// TIA Portal V21 export
FUNCTION "BOWIE" : Void   // FC7, LAD
{ S7_Optimized_Access := 'TRUE' }
// stored: SetENOAutomatically false
   VAR_TEMP
      START : Bool;
   END_VAR
   VAR_TEMP   // added for the SCL form of the ladder/FBD networks
      _w1 : Bool;
      _w2 : Bool;
      _w3 : Bool;
      _w4 : Bool;
   END_VAR
BEGIN

REGION Network 1
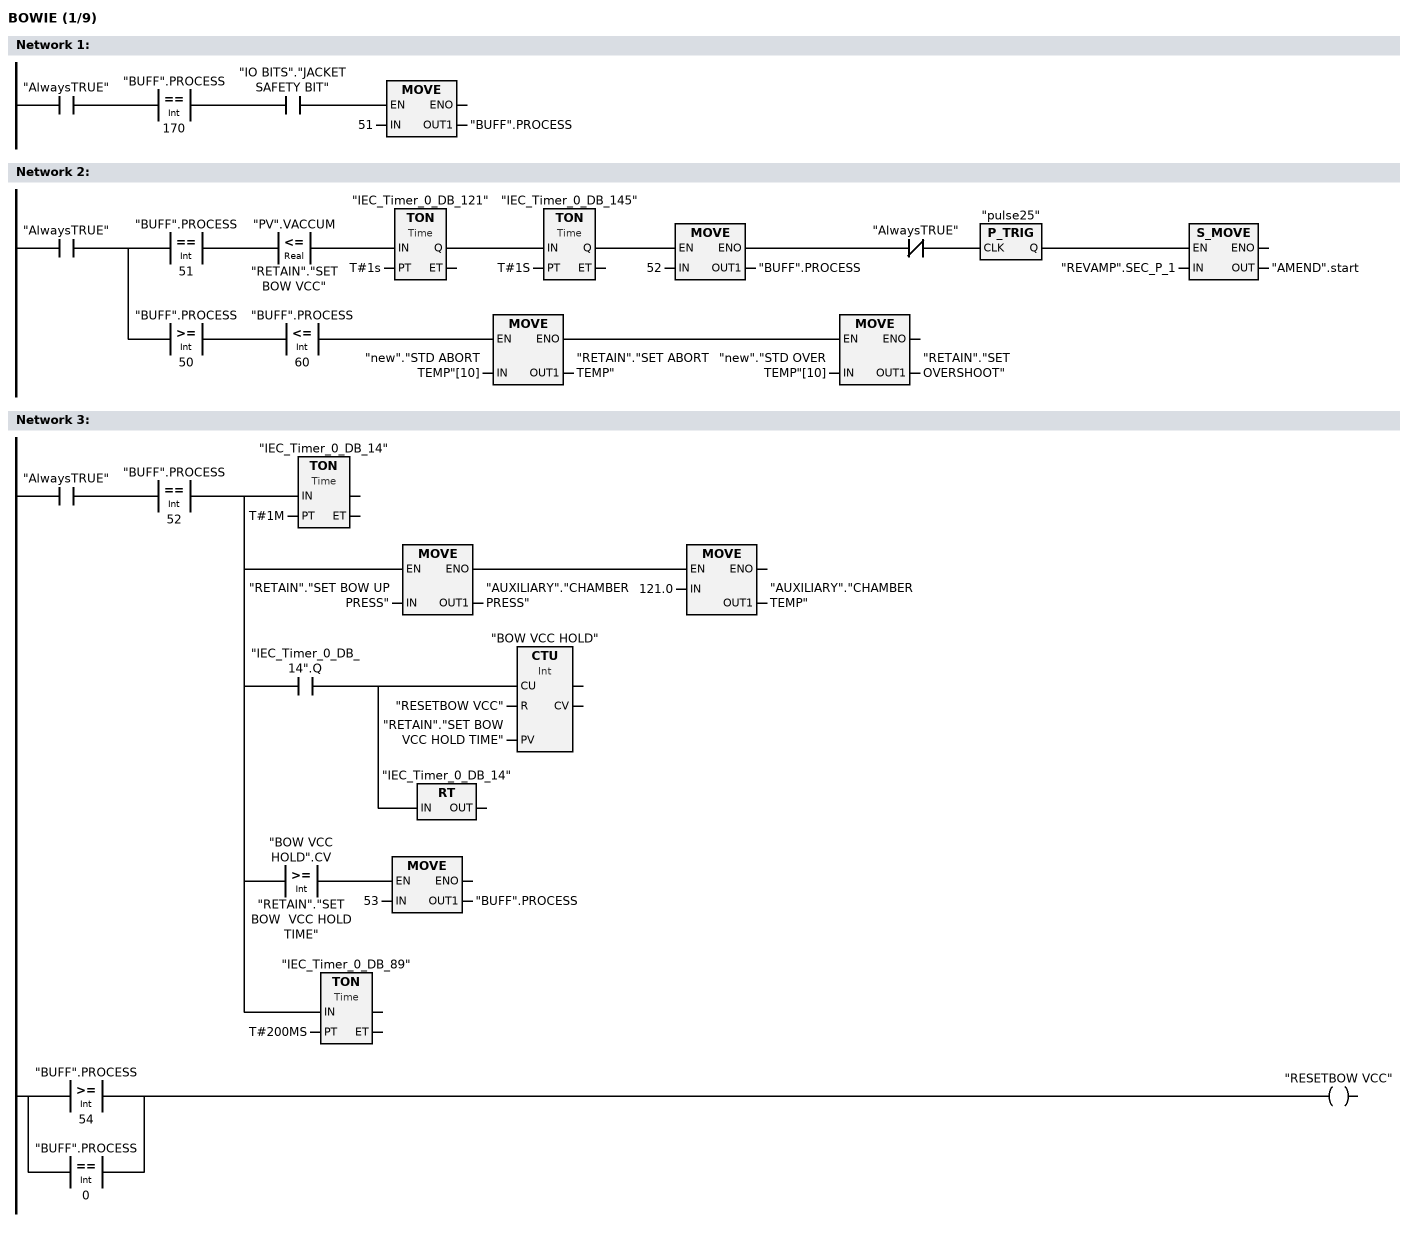
   RUNG wire#powerrail
      Contact( "AlwaysTRUE" )
      { S7_Templates := "SrcType := Int" } EQ_Contact(in1 := "BUFF".PROCESS, in2 := 170)
      Contact( "IO BITS"."JACKET SAFETY BIT" )
      Move(in := 51, out1 => "BUFF".PROCESS)
   END_RUNG
   // the same network as SCL:
   IF "AlwaysTRUE" AND ("BUFF".PROCESS = 170) AND "IO BITS"."JACKET SAFETY BIT" THEN
       "BUFF".PROCESS := 51;
   END_IF;
END_REGION

REGION Network 2
   RUNG wire#powerrail
      Contact( "AlwaysTRUE" )
      wire#w1
      { S7_Templates := "SrcType := Int" } EQ_Contact(in1 := "BUFF".PROCESS, in2 := 51)
      { S7_Templates := "SrcType := Real" } LE_Contact(in1 := "PV".VACCUM, in2 := "RETAIN"."SET BOW VCC")
      { S7_Templates := "time_type := Time" } "IEC_Timer_0_DB_121".TON(pt := T#1s, et =>)
      { S7_Templates := "time_type := Time" } "IEC_Timer_0_DB_145".TON(pt := T#1S, et =>)
      Move(in := 52, out1 => "BUFF".PROCESS)
      I_Contact( "AlwaysTRUE" )
      P_Trig( "pulse25" )
      S_Move(in := "REVAMP".SEC_P_1, out => "AMEND".start)
   END_RUNG
   RUNG wire#w1
      { S7_Templates := "SrcType := Int" } GE_Contact(in1 := "BUFF".PROCESS, in2 := 50)
      { S7_Templates := "SrcType := Int" } LE_Contact(in1 := "BUFF".PROCESS, in2 := 60)
      Move(in := "new"."STD ABORT TEMP"[10], out1 => "RETAIN"."SET ABORT TEMP")
      Move(in := "new"."STD OVER TEMP"[10], out1 => "RETAIN"."SET OVERSHOOT")
   END_RUNG
   // the same network as SCL:
   "IEC_Timer_0_DB_121".TON(IN := "AlwaysTRUE" AND ("BUFF".PROCESS = 51) AND ("PV".VACCUM <= "RETAIN"."SET BOW VCC"),
                           PT := T#1s);
   "IEC_Timer_0_DB_145".TON(IN := "IEC_Timer_0_DB_121".Q, PT := T#1S);
   IF "IEC_Timer_0_DB_145".Q THEN "BUFF".PROCESS := 52; END_IF;
   #_w1 := "IEC_Timer_0_DB_145".Q AND NOT "AlwaysTRUE";
   #_w2 := #_w1 AND NOT "pulse25";   // rising edge
   "pulse25" := #_w1;
   IF #_w2 THEN "AMEND".start := "REVAMP".SEC_P_1; END_IF;
   IF "AlwaysTRUE" AND ("BUFF".PROCESS >= 50) AND ("BUFF".PROCESS <= 60) THEN
       "RETAIN"."SET ABORT TEMP" := "new"."STD ABORT TEMP"[10];
       "RETAIN"."SET OVERSHOOT" := "new"."STD OVER TEMP"[10];
   END_IF;
END_REGION

REGION Network 3
   RUNG wire#powerrail
      Contact( "AlwaysTRUE" )
      { S7_Templates := "SrcType := Int" } EQ_Contact(in1 := "BUFF".PROCESS, in2 := 52)
      wire#w1
      { S7_Templates := "time_type := Time" } "IEC_Timer_0_DB_14".TON(pt := T#1M, et =>)
   END_RUNG
   RUNG wire#w1
      Move(in := "RETAIN"."SET BOW UP PRESS", out1 => "AUXILIARY"."CHAMBER PRESS")
      Move(in := 121.0, out1 => "AUXILIARY"."CHAMBER TEMP")
   END_RUNG
   RUNG wire#w1
      Contact( "IEC_Timer_0_DB_14".Q )
      wire#w2
      { S7_Templates := "value_type := Int" } "BOW VCC HOLD".CTU(r := "RESETBOW VCC", pv := "RETAIN"."SET BOW  VCC HOLD TIME", cv =>)
   END_RUNG
   RUNG wire#w2
      RT_Coil( "IEC_Timer_0_DB_14" )
   END_RUNG
   RUNG wire#w1
      { S7_Templates := "SrcType := Int" } GE_Contact(in1 := "BOW VCC HOLD".CV, in2 := "RETAIN"."SET BOW  VCC HOLD TIME")
      Move(in := 53, out1 => "BUFF".PROCESS)
   END_RUNG
   RUNG wire#w1
      { S7_Templates := "time_type := Time" } "IEC_Timer_0_DB_89".TON(pt := T#200MS, et =>)
   END_RUNG
   RUNG wire#powerrail
      { S7_Templates := "SrcType := Int" } GE_Contact(in1 := "BUFF".PROCESS, in2 := 54)
      wire#w3
      Coil( "RESETBOW VCC" )
   END_RUNG
   RUNG wire#powerrail
      { S7_Templates := "SrcType := Int" } EQ_Contact(in1 := "BUFF".PROCESS, in2 := 0)
   END_RUNG wire#w3
   // the same network as SCL:
   #_w1 := "AlwaysTRUE" AND ("BUFF".PROCESS = 52);
   "IEC_Timer_0_DB_14".TON(IN := #_w1, PT := T#1M);
   IF #_w1 THEN
       "AUXILIARY"."CHAMBER PRESS" := "RETAIN"."SET BOW UP PRESS";
       "AUXILIARY"."CHAMBER TEMP" := 121.0;
   END_IF;
   #_w2 := #_w1 AND "IEC_Timer_0_DB_14".Q;
   "BOW VCC HOLD".CTU(CU := #_w2, R := "RESETBOW VCC", PV := "RETAIN"."SET BOW  VCC HOLD TIME");
   IF #_w2 THEN RESET_TIMER("IEC_Timer_0_DB_14"); END_IF;
   IF #_w1 AND ("BOW VCC HOLD".CV >= "RETAIN"."SET BOW  VCC HOLD TIME") THEN "BUFF".PROCESS := 53; END_IF;
   "IEC_Timer_0_DB_89".TON(IN := #_w1, PT := T#200MS);
   "RESETBOW VCC" := ("BUFF".PROCESS >= 54) OR ("BUFF".PROCESS = 0);
END_REGION

REGION Network 4
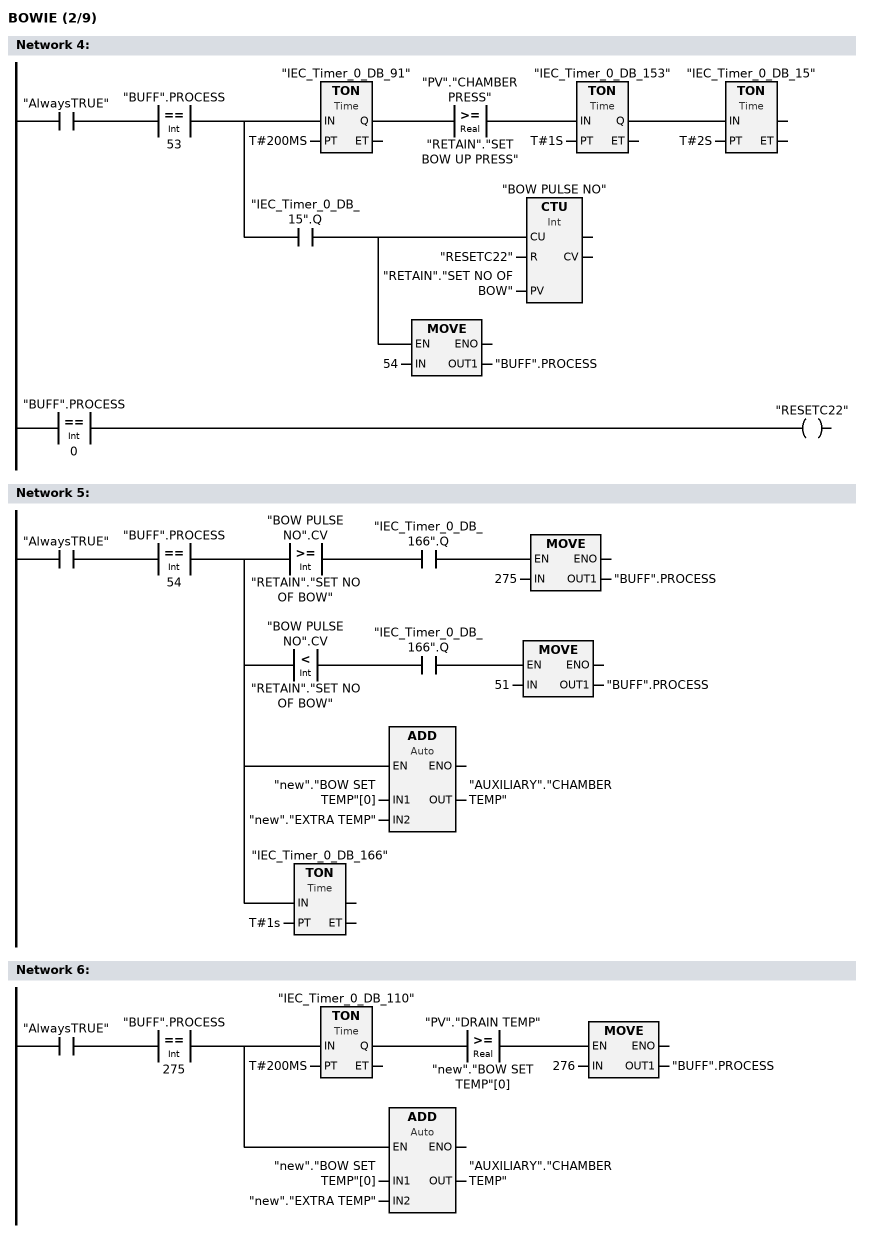
   RUNG wire#powerrail
      Contact( "AlwaysTRUE" )
      { S7_Templates := "SrcType := Int" } EQ_Contact(in1 := "BUFF".PROCESS, in2 := 53)
      wire#w1
      { S7_Templates := "time_type := Time" } "IEC_Timer_0_DB_91".TON(pt := T#200MS, et =>)
      { S7_Templates := "SrcType := Real" } GE_Contact(in1 := "PV"."CHAMBER PRESS", in2 := "RETAIN"."SET BOW UP PRESS")
      { S7_Templates := "time_type := Time" } "IEC_Timer_0_DB_153".TON(pt := T#1S, et =>)
      { S7_Templates := "time_type := Time" } "IEC_Timer_0_DB_15".TON(pt := T#2S, et =>)
   END_RUNG
   RUNG wire#w1
      Contact( "IEC_Timer_0_DB_15".Q )
      wire#w2
      { S7_Templates := "value_type := Int" } "BOW PULSE NO".CTU(r := "RESETC22", pv := "RETAIN"."SET NO OF BOW", cv =>)
   END_RUNG
   RUNG wire#w2
      Move(in := 54, out1 => "BUFF".PROCESS)
   END_RUNG
   RUNG wire#powerrail
      { S7_Templates := "SrcType := Int" } EQ_Contact(in1 := "BUFF".PROCESS, in2 := 0)
      Coil( "RESETC22" )
   END_RUNG
   // the same network as SCL:
   #_w1 := "AlwaysTRUE" AND ("BUFF".PROCESS = 53);
   "IEC_Timer_0_DB_91".TON(IN := #_w1, PT := T#200MS);
   "IEC_Timer_0_DB_153".TON(IN := "IEC_Timer_0_DB_91".Q AND ("PV"."CHAMBER PRESS" >= "RETAIN"."SET BOW UP PRESS"),
                           PT := T#1S);
   "IEC_Timer_0_DB_15".TON(IN := "IEC_Timer_0_DB_153".Q, PT := T#2S);
   #_w2 := #_w1 AND "IEC_Timer_0_DB_15".Q;
   "BOW PULSE NO".CTU(CU := #_w2, R := "RESETC22", PV := "RETAIN"."SET NO OF BOW");
   IF #_w2 THEN "BUFF".PROCESS := 54; END_IF;
   "RESETC22" := "BUFF".PROCESS = 0;
END_REGION

REGION Network 5
   RUNG wire#powerrail
      Contact( "AlwaysTRUE" )
      { S7_Templates := "SrcType := Int" } EQ_Contact(in1 := "BUFF".PROCESS, in2 := 54)
      wire#w1
      { S7_Templates := "SrcType := Int" } GE_Contact(in1 := "BOW PULSE NO".CV, in2 := "RETAIN"."SET NO OF BOW")
      Contact( "IEC_Timer_0_DB_166".Q )
      Move(in := 275, out1 => "BUFF".PROCESS)
   END_RUNG
   RUNG wire#w1
      { S7_Templates := "SrcType := Int" } LT_Contact(in1 := "BOW PULSE NO".CV, in2 := "RETAIN"."SET NO OF BOW")
      Contact( "IEC_Timer_0_DB_166".Q )
      Move(in := 51, out1 => "BUFF".PROCESS)
   END_RUNG
   RUNG wire#w1
      Add(in1 := "new"."BOW SET TEMP"[0], in2 := "new"."EXTRA TEMP", out => "AUXILIARY"."CHAMBER TEMP")
   END_RUNG
   RUNG wire#w1
      { S7_Templates := "time_type := Time" } "IEC_Timer_0_DB_166".TON(pt := T#1s, et =>)
   END_RUNG
   // the same network as SCL:
   #_w1 := "AlwaysTRUE" AND ("BUFF".PROCESS = 54);
   IF #_w1 AND ("BOW PULSE NO".CV >= "RETAIN"."SET NO OF BOW") AND "IEC_Timer_0_DB_166".Q THEN
       "BUFF".PROCESS := 275;
   END_IF;
   IF #_w1 AND ("BOW PULSE NO".CV < "RETAIN"."SET NO OF BOW") AND "IEC_Timer_0_DB_166".Q THEN
       "BUFF".PROCESS := 51;
   END_IF;
   IF #_w1 THEN "AUXILIARY"."CHAMBER TEMP" := "new"."BOW SET TEMP"[0] + "new"."EXTRA TEMP"; END_IF;
   "IEC_Timer_0_DB_166".TON(IN := #_w1, PT := T#1s);
END_REGION

REGION Network 6
   RUNG wire#powerrail
      Contact( "AlwaysTRUE" )
      { S7_Templates := "SrcType := Int" } EQ_Contact(in1 := "BUFF".PROCESS, in2 := 275)
      wire#w1
      { S7_Templates := "time_type := Time" } "IEC_Timer_0_DB_110".TON(pt := T#200MS, et =>)
      { S7_Templates := "SrcType := Real" } GE_Contact(in1 := "PV"."DRAIN TEMP", in2 := "new"."BOW SET TEMP"[0])
      Move(in := 276, out1 => "BUFF".PROCESS)
   END_RUNG
   RUNG wire#w1
      Add(in1 := "new"."BOW SET TEMP"[0], in2 := "new"."EXTRA TEMP", out => "AUXILIARY"."CHAMBER TEMP")
   END_RUNG
   // the same network as SCL:
   #_w1 := "AlwaysTRUE" AND ("BUFF".PROCESS = 275);
   "IEC_Timer_0_DB_110".TON(IN := #_w1, PT := T#200MS);
   IF "IEC_Timer_0_DB_110".Q AND ("PV"."DRAIN TEMP" >= "new"."BOW SET TEMP"[0]) THEN
       "BUFF".PROCESS := 276;
   END_IF;
   IF #_w1 THEN "AUXILIARY"."CHAMBER TEMP" := "new"."BOW SET TEMP"[0] + "new"."EXTRA TEMP"; END_IF;
END_REGION

REGION Network 7
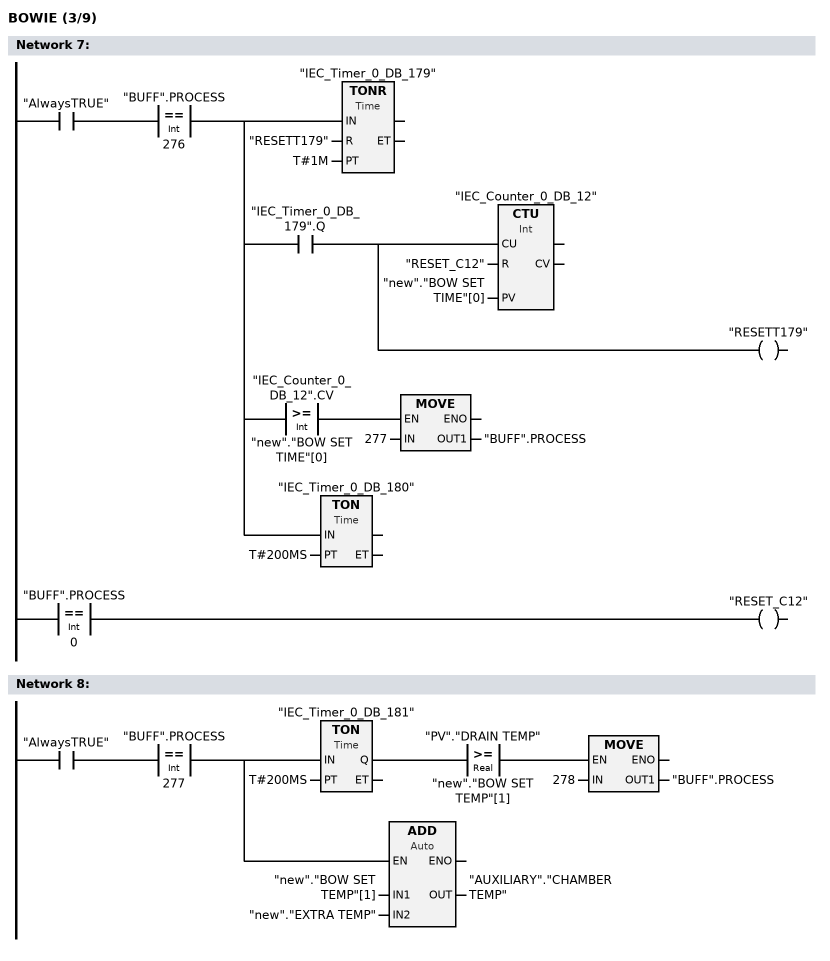
   RUNG wire#powerrail
      Contact( "AlwaysTRUE" )
      { S7_Templates := "SrcType := Int" } EQ_Contact(in1 := "BUFF".PROCESS, in2 := 276)
      wire#w1
      { S7_Templates := "time_type := Time" } "IEC_Timer_0_DB_179".TONR(r := "RESETT179", pt := T#1M, et =>)
   END_RUNG
   RUNG wire#w1
      Contact( "IEC_Timer_0_DB_179".Q )
      wire#w2
      { S7_Templates := "value_type := Int" } "IEC_Counter_0_DB_12".CTU(r := "RESET_C12", pv := "new"."BOW SET TIME"[0], cv =>)
   END_RUNG
   RUNG wire#w2
      Coil( "RESETT179" )
   END_RUNG
   RUNG wire#w1
      { S7_Templates := "SrcType := Int" } GE_Contact(in1 := "IEC_Counter_0_DB_12".CV, in2 := "new"."BOW SET TIME"[0])
      Move(in := 277, out1 => "BUFF".PROCESS)
   END_RUNG
   RUNG wire#w1
      { S7_Templates := "time_type := Time" } "IEC_Timer_0_DB_180".TON(pt := T#200MS, et =>)
   END_RUNG
   RUNG wire#powerrail
      { S7_Templates := "SrcType := Int" } EQ_Contact(in1 := "BUFF".PROCESS, in2 := 0)
      Coil( "RESET_C12" )
   END_RUNG
   // the same network as SCL:
   #_w1 := "AlwaysTRUE" AND ("BUFF".PROCESS = 276);
   "IEC_Timer_0_DB_179".TONR(IN := #_w1, R := "RESETT179", PT := T#1M);
   #_w2 := #_w1 AND "IEC_Timer_0_DB_179".Q;
   "IEC_Counter_0_DB_12".CTU(CU := #_w2, R := "RESET_C12", PV := "new"."BOW SET TIME"[0]);
   "RESETT179" := #_w2;
   IF #_w1 AND ("IEC_Counter_0_DB_12".CV >= "new"."BOW SET TIME"[0]) THEN "BUFF".PROCESS := 277; END_IF;
   "IEC_Timer_0_DB_180".TON(IN := #_w1, PT := T#200MS);
   "RESET_C12" := "BUFF".PROCESS = 0;
END_REGION

REGION Network 8
   RUNG wire#powerrail
      Contact( "AlwaysTRUE" )
      { S7_Templates := "SrcType := Int" } EQ_Contact(in1 := "BUFF".PROCESS, in2 := 277)
      wire#w1
      { S7_Templates := "time_type := Time" } "IEC_Timer_0_DB_181".TON(pt := T#200MS, et =>)
      { S7_Templates := "SrcType := Real" } GE_Contact(in1 := "PV"."DRAIN TEMP", in2 := "new"."BOW SET TEMP"[1])
      Move(in := 278, out1 => "BUFF".PROCESS)
   END_RUNG
   RUNG wire#w1
      Add(in1 := "new"."BOW SET TEMP"[1], in2 := "new"."EXTRA TEMP", out => "AUXILIARY"."CHAMBER TEMP")
   END_RUNG
   // the same network as SCL:
   #_w1 := "AlwaysTRUE" AND ("BUFF".PROCESS = 277);
   "IEC_Timer_0_DB_181".TON(IN := #_w1, PT := T#200MS);
   IF "IEC_Timer_0_DB_181".Q AND ("PV"."DRAIN TEMP" >= "new"."BOW SET TEMP"[1]) THEN
       "BUFF".PROCESS := 278;
   END_IF;
   IF #_w1 THEN "AUXILIARY"."CHAMBER TEMP" := "new"."BOW SET TEMP"[1] + "new"."EXTRA TEMP"; END_IF;
END_REGION

REGION Network 9
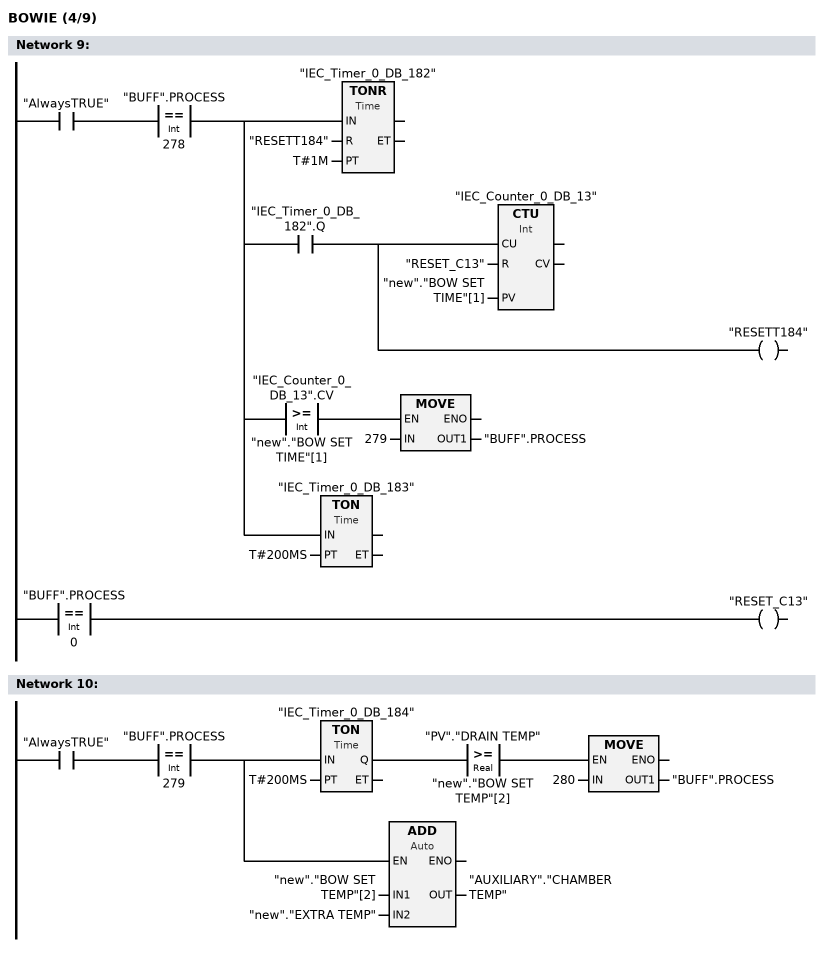
   RUNG wire#powerrail
      Contact( "AlwaysTRUE" )
      { S7_Templates := "SrcType := Int" } EQ_Contact(in1 := "BUFF".PROCESS, in2 := 278)
      wire#w1
      { S7_Templates := "time_type := Time" } "IEC_Timer_0_DB_182".TONR(r := "RESETT184", pt := T#1M, et =>)
   END_RUNG
   RUNG wire#w1
      Contact( "IEC_Timer_0_DB_182".Q )
      wire#w2
      { S7_Templates := "value_type := Int" } "IEC_Counter_0_DB_13".CTU(r := "RESET_C13", pv := "new"."BOW SET TIME"[1], cv =>)
   END_RUNG
   RUNG wire#w2
      Coil( "RESETT184" )
   END_RUNG
   RUNG wire#w1
      { S7_Templates := "SrcType := Int" } GE_Contact(in1 := "IEC_Counter_0_DB_13".CV, in2 := "new"."BOW SET TIME"[1])
      Move(in := 279, out1 => "BUFF".PROCESS)
   END_RUNG
   RUNG wire#w1
      { S7_Templates := "time_type := Time" } "IEC_Timer_0_DB_183".TON(pt := T#200MS, et =>)
   END_RUNG
   RUNG wire#powerrail
      { S7_Templates := "SrcType := Int" } EQ_Contact(in1 := "BUFF".PROCESS, in2 := 0)
      Coil( "RESET_C13" )
   END_RUNG
   // the same network as SCL:
   #_w1 := "AlwaysTRUE" AND ("BUFF".PROCESS = 278);
   "IEC_Timer_0_DB_182".TONR(IN := #_w1, R := "RESETT184", PT := T#1M);
   #_w2 := #_w1 AND "IEC_Timer_0_DB_182".Q;
   "IEC_Counter_0_DB_13".CTU(CU := #_w2, R := "RESET_C13", PV := "new"."BOW SET TIME"[1]);
   "RESETT184" := #_w2;
   IF #_w1 AND ("IEC_Counter_0_DB_13".CV >= "new"."BOW SET TIME"[1]) THEN "BUFF".PROCESS := 279; END_IF;
   "IEC_Timer_0_DB_183".TON(IN := #_w1, PT := T#200MS);
   "RESET_C13" := "BUFF".PROCESS = 0;
END_REGION

REGION Network 10
   RUNG wire#powerrail
      Contact( "AlwaysTRUE" )
      { S7_Templates := "SrcType := Int" } EQ_Contact(in1 := "BUFF".PROCESS, in2 := 279)
      wire#w1
      { S7_Templates := "time_type := Time" } "IEC_Timer_0_DB_184".TON(pt := T#200MS, et =>)
      { S7_Templates := "SrcType := Real" } GE_Contact(in1 := "PV"."DRAIN TEMP", in2 := "new"."BOW SET TEMP"[2])
      Move(in := 280, out1 => "BUFF".PROCESS)
   END_RUNG
   RUNG wire#w1
      Add(in1 := "new"."BOW SET TEMP"[2], in2 := "new"."EXTRA TEMP", out => "AUXILIARY"."CHAMBER TEMP")
   END_RUNG
   // the same network as SCL:
   #_w1 := "AlwaysTRUE" AND ("BUFF".PROCESS = 279);
   "IEC_Timer_0_DB_184".TON(IN := #_w1, PT := T#200MS);
   IF "IEC_Timer_0_DB_184".Q AND ("PV"."DRAIN TEMP" >= "new"."BOW SET TEMP"[2]) THEN
       "BUFF".PROCESS := 280;
   END_IF;
   IF #_w1 THEN "AUXILIARY"."CHAMBER TEMP" := "new"."BOW SET TEMP"[2] + "new"."EXTRA TEMP"; END_IF;
END_REGION

REGION Network 11
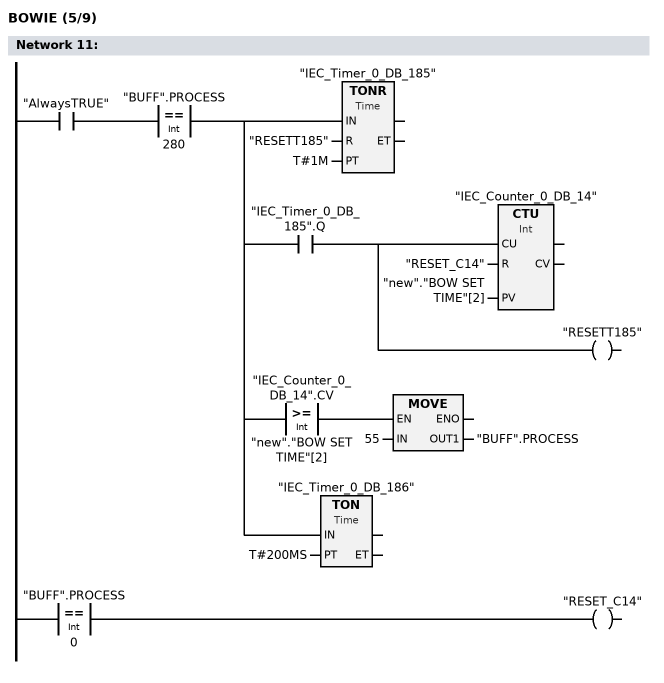
   RUNG wire#powerrail
      Contact( "AlwaysTRUE" )
      { S7_Templates := "SrcType := Int" } EQ_Contact(in1 := "BUFF".PROCESS, in2 := 280)
      wire#w1
      { S7_Templates := "time_type := Time" } "IEC_Timer_0_DB_185".TONR(r := "RESETT185", pt := T#1M, et =>)
   END_RUNG
   RUNG wire#w1
      Contact( "IEC_Timer_0_DB_185".Q )
      wire#w2
      { S7_Templates := "value_type := Int" } "IEC_Counter_0_DB_14".CTU(r := "RESET_C14", pv := "new"."BOW SET TIME"[2], cv =>)
   END_RUNG
   RUNG wire#w2
      Coil( "RESETT185" )
   END_RUNG
   RUNG wire#w1
      { S7_Templates := "SrcType := Int" } GE_Contact(in1 := "IEC_Counter_0_DB_14".CV, in2 := "new"."BOW SET TIME"[2])
      Move(in := 55, out1 => "BUFF".PROCESS)
   END_RUNG
   RUNG wire#w1
      { S7_Templates := "time_type := Time" } "IEC_Timer_0_DB_186".TON(pt := T#200MS, et =>)
   END_RUNG
   RUNG wire#powerrail
      { S7_Templates := "SrcType := Int" } EQ_Contact(in1 := "BUFF".PROCESS, in2 := 0)
      Coil( "RESET_C14" )
   END_RUNG
   // the same network as SCL:
   #_w1 := "AlwaysTRUE" AND ("BUFF".PROCESS = 280);
   "IEC_Timer_0_DB_185".TONR(IN := #_w1, R := "RESETT185", PT := T#1M);
   #_w2 := #_w1 AND "IEC_Timer_0_DB_185".Q;
   "IEC_Counter_0_DB_14".CTU(CU := #_w2, R := "RESET_C14", PV := "new"."BOW SET TIME"[2]);
   "RESETT185" := #_w2;
   IF #_w1 AND ("IEC_Counter_0_DB_14".CV >= "new"."BOW SET TIME"[2]) THEN "BUFF".PROCESS := 55; END_IF;
   "IEC_Timer_0_DB_186".TON(IN := #_w1, PT := T#200MS);
   "RESET_C14" := "BUFF".PROCESS = 0;
END_REGION

REGION Network 12
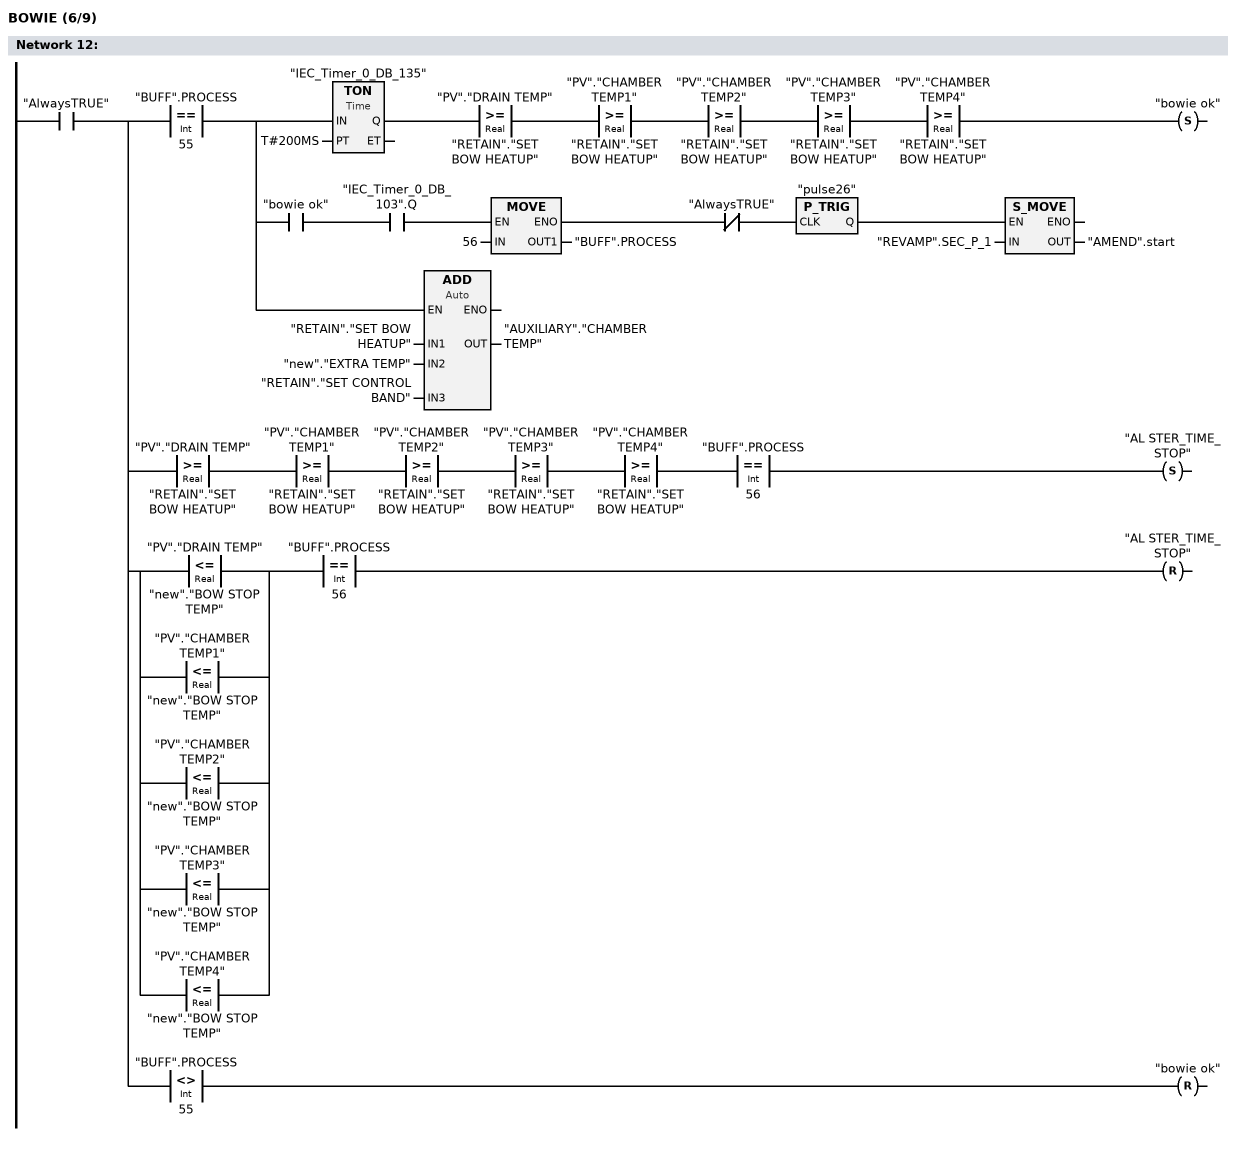
   RUNG wire#powerrail
      Contact( "AlwaysTRUE" )
      wire#w1
      { S7_Templates := "SrcType := Int" } EQ_Contact(in1 := "BUFF".PROCESS, in2 := 55)
      wire#w2
      { S7_Templates := "time_type := Time" } "IEC_Timer_0_DB_135".TON(pt := T#200MS, et =>)
      { S7_Templates := "SrcType := Real" } GE_Contact(in1 := "PV"."DRAIN TEMP", in2 := "RETAIN"."SET BOW HEATUP")
      { S7_Templates := "SrcType := Real" } GE_Contact(in1 := "PV"."CHAMBER TEMP1", in2 := "RETAIN"."SET BOW HEATUP")
      { S7_Templates := "SrcType := Real" } GE_Contact(in1 := "PV"."CHAMBER TEMP2", in2 := "RETAIN"."SET BOW HEATUP")
      { S7_Templates := "SrcType := Real" } GE_Contact(in1 := "PV"."CHAMBER TEMP3", in2 := "RETAIN"."SET BOW HEATUP")
      { S7_Templates := "SrcType := Real" } GE_Contact(in1 := "PV"."CHAMBER TEMP4", in2 := "RETAIN"."SET BOW HEATUP")
      S_Coil( "bowie ok" )
   END_RUNG
   RUNG wire#w2
      Contact( "bowie ok" )
      Contact( "IEC_Timer_0_DB_103".Q )
      Move(in := 56, out1 => "BUFF".PROCESS)
      I_Contact( "AlwaysTRUE" )
      P_Trig( "pulse26" )
      S_Move(in := "REVAMP".SEC_P_1, out => "AMEND".start)
   END_RUNG
   RUNG wire#w2
      Add(in1 := "RETAIN"."SET BOW HEATUP", in2 := "new"."EXTRA TEMP", in3 := "RETAIN"."SET CONTROL BAND", out => "AUXILIARY"."CHAMBER TEMP")
   END_RUNG
   RUNG wire#w1
      { S7_Templates := "SrcType := Real" } GE_Contact(in1 := "PV"."DRAIN TEMP", in2 := "RETAIN"."SET BOW HEATUP")
      { S7_Templates := "SrcType := Real" } GE_Contact(in1 := "PV"."CHAMBER TEMP1", in2 := "RETAIN"."SET BOW HEATUP")
      { S7_Templates := "SrcType := Real" } GE_Contact(in1 := "PV"."CHAMBER TEMP2", in2 := "RETAIN"."SET BOW HEATUP")
      { S7_Templates := "SrcType := Real" } GE_Contact(in1 := "PV"."CHAMBER TEMP3", in2 := "RETAIN"."SET BOW HEATUP")
      { S7_Templates := "SrcType := Real" } GE_Contact(in1 := "PV"."CHAMBER TEMP4", in2 := "RETAIN"."SET BOW HEATUP")
      { S7_Templates := "SrcType := Int" } EQ_Contact(in1 := "BUFF".PROCESS, in2 := 56)
      S_Coil( "AL STER_TIME_STOP" )
   END_RUNG
   RUNG wire#w1
      { S7_Templates := "SrcType := Real" } LE_Contact(in1 := "PV"."DRAIN TEMP", in2 := "new"."BOW STOP TEMP")
      wire#w3
      { S7_Templates := "SrcType := Int" } EQ_Contact(in1 := "BUFF".PROCESS, in2 := 56)
      R_Coil( "AL STER_TIME_STOP" )
   END_RUNG
   RUNG wire#w1
      { S7_Templates := "SrcType := Real" } LE_Contact(in1 := "PV"."CHAMBER TEMP1", in2 := "new"."BOW STOP TEMP")
   END_RUNG wire#w3
   RUNG wire#w1
      { S7_Templates := "SrcType := Real" } LE_Contact(in1 := "PV"."CHAMBER TEMP2", in2 := "new"."BOW STOP TEMP")
   END_RUNG wire#w3
   RUNG wire#w1
      { S7_Templates := "SrcType := Real" } LE_Contact(in1 := "PV"."CHAMBER TEMP3", in2 := "new"."BOW STOP TEMP")
   END_RUNG wire#w3
   RUNG wire#w1
      { S7_Templates := "SrcType := Real" } LE_Contact(in1 := "PV"."CHAMBER TEMP4", in2 := "new"."BOW STOP TEMP")
   END_RUNG wire#w3
   RUNG wire#w1
      { S7_Templates := "SrcType := Int" } NE_Contact(in1 := "BUFF".PROCESS, in2 := 55)
      R_Coil( "bowie ok" )
   END_RUNG
   // the same network as SCL:
   #_w1 := "AlwaysTRUE" AND ("BUFF".PROCESS = 55);
   "IEC_Timer_0_DB_135".TON(IN := #_w1, PT := T#200MS);
   IF "IEC_Timer_0_DB_135".Q AND ("PV"."DRAIN TEMP" >= "RETAIN"."SET BOW HEATUP") AND ("PV"."CHAMBER TEMP1" >= "RETAIN"."SET BOW HEATUP") AND ("PV"."CHAMBER TEMP2" >= "RETAIN"."SET BOW HEATUP") AND ("PV"."CHAMBER TEMP3" >= "RETAIN"."SET BOW HEATUP") AND ("PV"."CHAMBER TEMP4" >= "RETAIN"."SET BOW HEATUP") THEN
       "bowie ok" := TRUE;
   END_IF;
   #_w2 := #_w1 AND "bowie ok" AND "IEC_Timer_0_DB_103".Q;
   IF #_w2 THEN "BUFF".PROCESS := 56; END_IF;
   #_w3 := #_w2 AND NOT "AlwaysTRUE";
   #_w4 := #_w3 AND NOT "pulse26";   // rising edge
   "pulse26" := #_w3;
   IF #_w4 THEN "AMEND".start := "REVAMP".SEC_P_1; END_IF;
   IF #_w1 THEN
       "AUXILIARY"."CHAMBER TEMP" := "RETAIN"."SET BOW HEATUP" + "new"."EXTRA TEMP" + "RETAIN"."SET CONTROL BAND";
   END_IF;
   IF "AlwaysTRUE" AND ("PV"."DRAIN TEMP" >= "RETAIN"."SET BOW HEATUP") AND ("PV"."CHAMBER TEMP1" >= "RETAIN"."SET BOW HEATUP") AND ("PV"."CHAMBER TEMP2" >= "RETAIN"."SET BOW HEATUP") AND ("PV"."CHAMBER TEMP3" >= "RETAIN"."SET BOW HEATUP") AND ("PV"."CHAMBER TEMP4" >= "RETAIN"."SET BOW HEATUP") AND ("BUFF".PROCESS = 56) THEN
       "AL STER_TIME_STOP" := TRUE;
   END_IF;
   IF "AlwaysTRUE" AND (("PV"."DRAIN TEMP" <= "new"."BOW STOP TEMP") OR ("PV"."CHAMBER TEMP1" <= "new"."BOW STOP TEMP") OR ("PV"."CHAMBER TEMP2" <= "new"."BOW STOP TEMP") OR ("PV"."CHAMBER TEMP3" <= "new"."BOW STOP TEMP") OR ("PV"."CHAMBER TEMP4" <= "new"."BOW STOP TEMP")) AND ("BUFF".PROCESS = 56) THEN
       "AL STER_TIME_STOP" := FALSE;
   END_IF;
   IF "AlwaysTRUE" AND ("BUFF".PROCESS <> 55) THEN "bowie ok" := FALSE; END_IF;
END_REGION

REGION Network 13
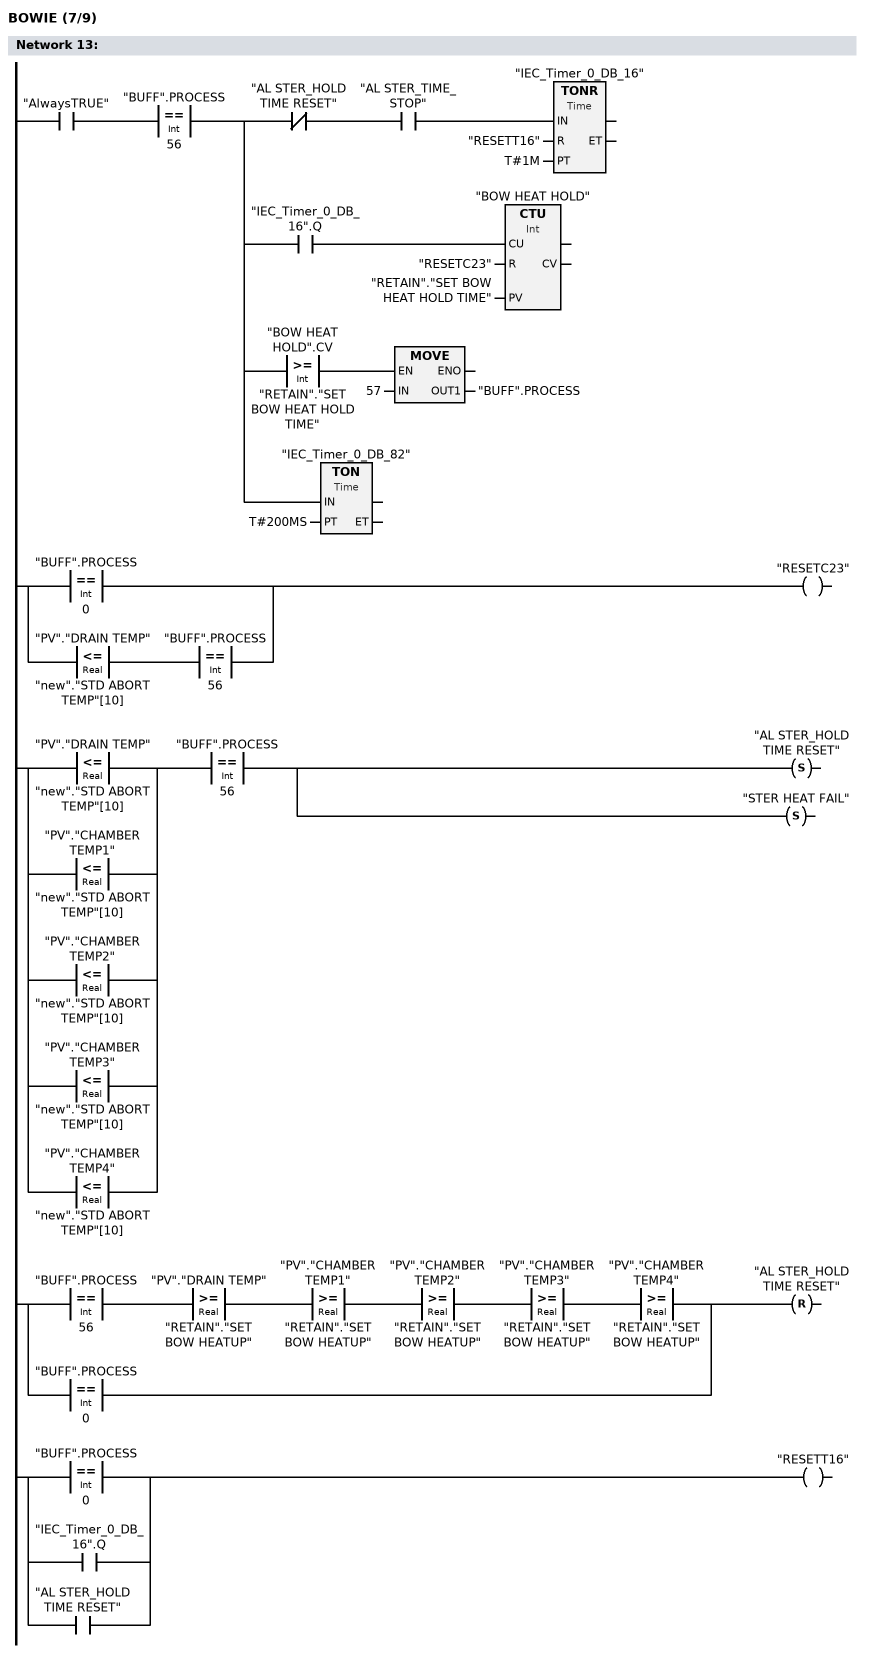
   RUNG wire#powerrail
      Contact( "AlwaysTRUE" )
      { S7_Templates := "SrcType := Int" } EQ_Contact(in1 := "BUFF".PROCESS, in2 := 56)
      wire#w1
      I_Contact( "AL STER_HOLD TIME RESET" )
      Contact( "AL STER_TIME_STOP" )
      { S7_Templates := "time_type := Time" } "IEC_Timer_0_DB_16".TONR(r := "RESETT16", pt := T#1M, et =>)
   END_RUNG
   RUNG wire#w1
      Contact( "IEC_Timer_0_DB_16".Q )
      { S7_Templates := "value_type := Int" } "BOW HEAT HOLD".CTU(r := "RESETC23", pv := "RETAIN"."SET BOW HEAT HOLD TIME", cv =>)
   END_RUNG
   RUNG wire#w1
      { S7_Templates := "SrcType := Int" } GE_Contact(in1 := "BOW HEAT HOLD".CV, in2 := "RETAIN"."SET BOW HEAT HOLD TIME")
      Move(in := 57, out1 => "BUFF".PROCESS)
   END_RUNG
   RUNG wire#w1
      { S7_Templates := "time_type := Time" } "IEC_Timer_0_DB_82".TON(pt := T#200MS, et =>)
   END_RUNG
   RUNG wire#powerrail
      { S7_Templates := "SrcType := Int" } EQ_Contact(in1 := "BUFF".PROCESS, in2 := 0)
      wire#w2
      Coil( "RESETC23" )
   END_RUNG
   RUNG wire#powerrail
      { S7_Templates := "SrcType := Real" } LE_Contact(in1 := "PV"."DRAIN TEMP", in2 := "new"."STD ABORT TEMP"[10])
      { S7_Templates := "SrcType := Int" } EQ_Contact(in1 := "BUFF".PROCESS, in2 := 56)
   END_RUNG wire#w2
   RUNG wire#powerrail
      { S7_Templates := "SrcType := Real" } LE_Contact(in1 := "PV"."DRAIN TEMP", in2 := "new"."STD ABORT TEMP"[10])
      wire#w3
      { S7_Templates := "SrcType := Int" } EQ_Contact(in1 := "BUFF".PROCESS, in2 := 56)
      wire#w4
      S_Coil( "AL STER_HOLD TIME RESET" )
   END_RUNG
   RUNG wire#powerrail
      { S7_Templates := "SrcType := Real" } LE_Contact(in1 := "PV"."CHAMBER TEMP1", in2 := "new"."STD ABORT TEMP"[10])
   END_RUNG wire#w3
   RUNG wire#powerrail
      { S7_Templates := "SrcType := Real" } LE_Contact(in1 := "PV"."CHAMBER TEMP2", in2 := "new"."STD ABORT TEMP"[10])
   END_RUNG wire#w3
   RUNG wire#powerrail
      { S7_Templates := "SrcType := Real" } LE_Contact(in1 := "PV"."CHAMBER TEMP3", in2 := "new"."STD ABORT TEMP"[10])
   END_RUNG wire#w3
   RUNG wire#powerrail
      { S7_Templates := "SrcType := Real" } LE_Contact(in1 := "PV"."CHAMBER TEMP4", in2 := "new"."STD ABORT TEMP"[10])
   END_RUNG wire#w3
   RUNG wire#w4
      S_Coil( "STER HEAT FAIL" )
   END_RUNG
   RUNG wire#powerrail
      { S7_Templates := "SrcType := Int" } EQ_Contact(in1 := "BUFF".PROCESS, in2 := 56)
      { S7_Templates := "SrcType := Real" } GE_Contact(in1 := "PV"."DRAIN TEMP", in2 := "RETAIN"."SET BOW HEATUP")
      { S7_Templates := "SrcType := Real" } GE_Contact(in1 := "PV"."CHAMBER TEMP1", in2 := "RETAIN"."SET BOW HEATUP")
      { S7_Templates := "SrcType := Real" } GE_Contact(in1 := "PV"."CHAMBER TEMP2", in2 := "RETAIN"."SET BOW HEATUP")
      { S7_Templates := "SrcType := Real" } GE_Contact(in1 := "PV"."CHAMBER TEMP3", in2 := "RETAIN"."SET BOW HEATUP")
      { S7_Templates := "SrcType := Real" } GE_Contact(in1 := "PV"."CHAMBER TEMP4", in2 := "RETAIN"."SET BOW HEATUP")
      wire#w5
      R_Coil( "AL STER_HOLD TIME RESET" )
   END_RUNG
   RUNG wire#powerrail
      { S7_Templates := "SrcType := Int" } EQ_Contact(in1 := "BUFF".PROCESS, in2 := 0)
   END_RUNG wire#w5
   RUNG wire#powerrail
      { S7_Templates := "SrcType := Int" } EQ_Contact(in1 := "BUFF".PROCESS, in2 := 0)
      wire#w6
      Coil( "RESETT16" )
   END_RUNG
   RUNG wire#powerrail
      Contact( "IEC_Timer_0_DB_16".Q )
   END_RUNG wire#w6
   RUNG wire#powerrail
      Contact( "AL STER_HOLD TIME RESET" )
   END_RUNG wire#w6
   // the same network as SCL:
   #_w1 := "AlwaysTRUE" AND ("BUFF".PROCESS = 56);
   "IEC_Timer_0_DB_16".TONR(IN := #_w1 AND NOT "AL STER_HOLD TIME RESET" AND "AL STER_TIME_STOP",
                           R := "RESETT16",
                           PT := T#1M);
   "BOW HEAT HOLD".CTU(CU := #_w1 AND "IEC_Timer_0_DB_16".Q,
                       R := "RESETC23",
                       PV := "RETAIN"."SET BOW HEAT HOLD TIME");
   IF #_w1 AND ("BOW HEAT HOLD".CV >= "RETAIN"."SET BOW HEAT HOLD TIME") THEN "BUFF".PROCESS := 57; END_IF;
   "IEC_Timer_0_DB_82".TON(IN := #_w1, PT := T#200MS);
   "RESETC23" := ("BUFF".PROCESS = 0) OR (("PV"."DRAIN TEMP" <= "new"."STD ABORT TEMP"[10]) AND ("BUFF".PROCESS = 56));
   IF (("PV"."DRAIN TEMP" <= "new"."STD ABORT TEMP"[10]) OR ("PV"."CHAMBER TEMP1" <= "new"."STD ABORT TEMP"[10]) OR ("PV"."CHAMBER TEMP2" <= "new"."STD ABORT TEMP"[10]) OR ("PV"."CHAMBER TEMP3" <= "new"."STD ABORT TEMP"[10]) OR ("PV"."CHAMBER TEMP4" <= "new"."STD ABORT TEMP"[10])) AND ("BUFF".PROCESS = 56) THEN
       "AL STER_HOLD TIME RESET" := TRUE;
       "STER HEAT FAIL" := TRUE;
   END_IF;
   IF (("BUFF".PROCESS = 56) AND ("PV"."DRAIN TEMP" >= "RETAIN"."SET BOW HEATUP") AND ("PV"."CHAMBER TEMP1" >= "RETAIN"."SET BOW HEATUP") AND ("PV"."CHAMBER TEMP2" >= "RETAIN"."SET BOW HEATUP") AND ("PV"."CHAMBER TEMP3" >= "RETAIN"."SET BOW HEATUP") AND ("PV"."CHAMBER TEMP4" >= "RETAIN"."SET BOW HEATUP")) OR ("BUFF".PROCESS = 0) THEN
       "AL STER_HOLD TIME RESET" := FALSE;
   END_IF;
   "RESETT16" := ("BUFF".PROCESS = 0) OR "IEC_Timer_0_DB_16".Q OR "AL STER_HOLD TIME RESET";
END_REGION

REGION Network 14
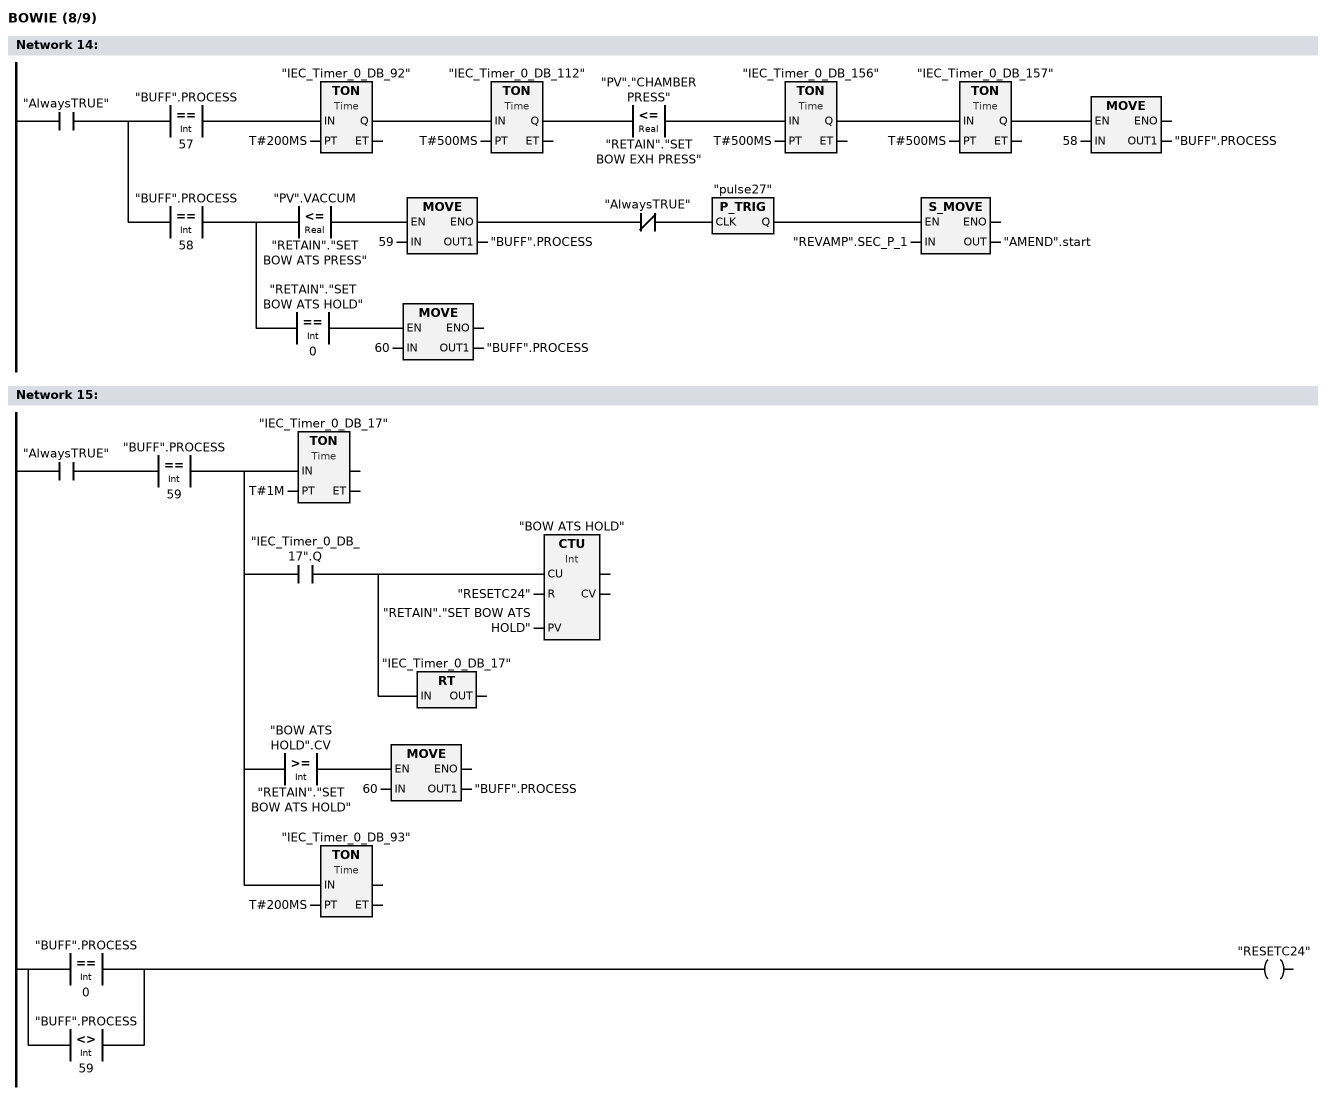
   RUNG wire#powerrail
      Contact( "AlwaysTRUE" )
      wire#w1
      { S7_Templates := "SrcType := Int" } EQ_Contact(in1 := "BUFF".PROCESS, in2 := 57)
      { S7_Templates := "time_type := Time" } "IEC_Timer_0_DB_92".TON(pt := T#200MS, et =>)
      { S7_Templates := "time_type := Time" } "IEC_Timer_0_DB_112".TON(pt := T#500MS, et =>)
      { S7_Templates := "SrcType := Real" } LE_Contact(in1 := "PV"."CHAMBER PRESS", in2 := "RETAIN"."SET BOW EXH PRESS")
      { S7_Templates := "time_type := Time" } "IEC_Timer_0_DB_156".TON(pt := T#500MS, et =>)
      { S7_Templates := "time_type := Time" } "IEC_Timer_0_DB_157".TON(pt := T#500MS, et =>)
      Move(in := 58, out1 => "BUFF".PROCESS)
   END_RUNG
   RUNG wire#w1
      { S7_Templates := "SrcType := Int" } EQ_Contact(in1 := "BUFF".PROCESS, in2 := 58)
      wire#w2
      { S7_Templates := "SrcType := Real" } LE_Contact(in1 := "PV".VACCUM, in2 := "RETAIN"."SET BOW ATS PRESS")
      Move(in := 59, out1 => "BUFF".PROCESS)
      I_Contact( "AlwaysTRUE" )
      P_Trig( "pulse27" )
      S_Move(in := "REVAMP".SEC_P_1, out => "AMEND".start)
   END_RUNG
   RUNG wire#w2
      { S7_Templates := "SrcType := Int" } EQ_Contact(in1 := "RETAIN"."SET BOW ATS HOLD", in2 := 0)
      Move(in := 60, out1 => "BUFF".PROCESS)
   END_RUNG
   // the same network as SCL:
   "IEC_Timer_0_DB_92".TON(IN := "AlwaysTRUE" AND ("BUFF".PROCESS = 57), PT := T#200MS);
   "IEC_Timer_0_DB_112".TON(IN := "IEC_Timer_0_DB_92".Q, PT := T#500MS);
   "IEC_Timer_0_DB_156".TON(IN := "IEC_Timer_0_DB_112".Q AND ("PV"."CHAMBER PRESS" <= "RETAIN"."SET BOW EXH PRESS"),
                           PT := T#500MS);
   "IEC_Timer_0_DB_157".TON(IN := "IEC_Timer_0_DB_156".Q, PT := T#500MS);
   IF "IEC_Timer_0_DB_157".Q THEN "BUFF".PROCESS := 58; END_IF;
   #_w1 := "AlwaysTRUE" AND ("BUFF".PROCESS = 58);
   #_w2 := #_w1 AND ("PV".VACCUM <= "RETAIN"."SET BOW ATS PRESS");
   IF #_w2 THEN "BUFF".PROCESS := 59; END_IF;
   #_w3 := #_w2 AND NOT "AlwaysTRUE";
   #_w4 := #_w3 AND NOT "pulse27";   // rising edge
   "pulse27" := #_w3;
   IF #_w4 THEN "AMEND".start := "REVAMP".SEC_P_1; END_IF;
   IF #_w1 AND ("RETAIN"."SET BOW ATS HOLD" = 0) THEN "BUFF".PROCESS := 60; END_IF;
END_REGION

REGION Network 15
   RUNG wire#powerrail
      Contact( "AlwaysTRUE" )
      { S7_Templates := "SrcType := Int" } EQ_Contact(in1 := "BUFF".PROCESS, in2 := 59)
      wire#w1
      { S7_Templates := "time_type := Time" } "IEC_Timer_0_DB_17".TON(pt := T#1M, et =>)
   END_RUNG
   RUNG wire#w1
      Contact( "IEC_Timer_0_DB_17".Q )
      wire#w2
      { S7_Templates := "value_type := Int" } "BOW ATS HOLD".CTU(r := "RESETC24", pv := "RETAIN"."SET BOW ATS HOLD", cv =>)
   END_RUNG
   RUNG wire#w2
      RT_Coil( "IEC_Timer_0_DB_17" )
   END_RUNG
   RUNG wire#w1
      { S7_Templates := "SrcType := Int" } GE_Contact(in1 := "BOW ATS HOLD".CV, in2 := "RETAIN"."SET BOW ATS HOLD")
      Move(in := 60, out1 => "BUFF".PROCESS)
   END_RUNG
   RUNG wire#w1
      { S7_Templates := "time_type := Time" } "IEC_Timer_0_DB_93".TON(pt := T#200MS, et =>)
   END_RUNG
   RUNG wire#powerrail
      { S7_Templates := "SrcType := Int" } EQ_Contact(in1 := "BUFF".PROCESS, in2 := 0)
      wire#w3
      Coil( "RESETC24" )
   END_RUNG
   RUNG wire#powerrail
      { S7_Templates := "SrcType := Int" } NE_Contact(in1 := "BUFF".PROCESS, in2 := 59)
   END_RUNG wire#w3
   // the same network as SCL:
   #_w1 := "AlwaysTRUE" AND ("BUFF".PROCESS = 59);
   "IEC_Timer_0_DB_17".TON(IN := #_w1, PT := T#1M);
   #_w2 := #_w1 AND "IEC_Timer_0_DB_17".Q;
   "BOW ATS HOLD".CTU(CU := #_w2, R := "RESETC24", PV := "RETAIN"."SET BOW ATS HOLD");
   IF #_w2 THEN RESET_TIMER("IEC_Timer_0_DB_17"); END_IF;
   IF #_w1 AND ("BOW ATS HOLD".CV >= "RETAIN"."SET BOW ATS HOLD") THEN "BUFF".PROCESS := 60; END_IF;
   "IEC_Timer_0_DB_93".TON(IN := #_w1, PT := T#200MS);
   "RESETC24" := ("BUFF".PROCESS = 0) OR ("BUFF".PROCESS <> 59);
END_REGION

REGION Network 16
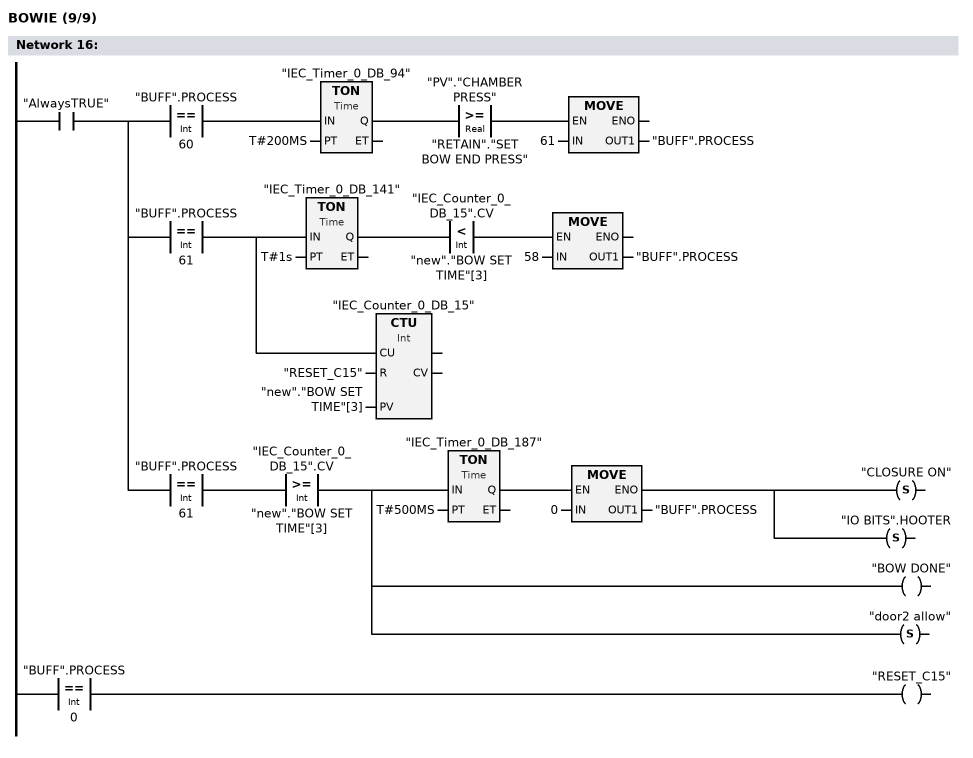
   RUNG wire#powerrail
      Contact( "AlwaysTRUE" )
      wire#w1
      { S7_Templates := "SrcType := Int" } EQ_Contact(in1 := "BUFF".PROCESS, in2 := 60)
      { S7_Templates := "time_type := Time" } "IEC_Timer_0_DB_94".TON(pt := T#200MS, et =>)
      { S7_Templates := "SrcType := Real" } GE_Contact(in1 := "PV"."CHAMBER PRESS", in2 := "RETAIN"."SET BOW END PRESS")
      Move(in := 61, out1 => "BUFF".PROCESS)
   END_RUNG
   RUNG wire#w1
      { S7_Templates := "SrcType := Int" } EQ_Contact(in1 := "BUFF".PROCESS, in2 := 61)
      wire#w2
      { S7_Templates := "time_type := Time" } "IEC_Timer_0_DB_141".TON(pt := T#1s, et =>)
      { S7_Templates := "SrcType := Int" } LT_Contact(in1 := "IEC_Counter_0_DB_15".CV, in2 := "new"."BOW SET TIME"[3])
      Move(in := 58, out1 => "BUFF".PROCESS)
   END_RUNG
   RUNG wire#w2
      { S7_Templates := "value_type := Int" } "IEC_Counter_0_DB_15".CTU(r := "RESET_C15", pv := "new"."BOW SET TIME"[3], cv =>)
   END_RUNG
   RUNG wire#w1
      { S7_Templates := "SrcType := Int" } EQ_Contact(in1 := "BUFF".PROCESS, in2 := 61)
      { S7_Templates := "SrcType := Int" } GE_Contact(in1 := "IEC_Counter_0_DB_15".CV, in2 := "new"."BOW SET TIME"[3])
      wire#w3
      { S7_Templates := "time_type := Time" } "IEC_Timer_0_DB_187".TON(pt := T#500MS, et =>)
      Move(in := 0, out1 => "BUFF".PROCESS)
      wire#w4
      S_Coil( "CLOSURE ON" )
   END_RUNG
   RUNG wire#w4
      S_Coil( "IO BITS".HOOTER )
   END_RUNG
   RUNG wire#w3
      Coil( "BOW DONE" )
   END_RUNG
   RUNG wire#w3
      S_Coil( "door2 allow" )
   END_RUNG
   RUNG wire#powerrail
      { S7_Templates := "SrcType := Int" } EQ_Contact(in1 := "BUFF".PROCESS, in2 := 0)
      Coil( "RESET_C15" )
   END_RUNG
   // the same network as SCL:
   "IEC_Timer_0_DB_94".TON(IN := "AlwaysTRUE" AND ("BUFF".PROCESS = 60), PT := T#200MS);
   IF "IEC_Timer_0_DB_94".Q AND ("PV"."CHAMBER PRESS" >= "RETAIN"."SET BOW END PRESS") THEN
       "BUFF".PROCESS := 61;
   END_IF;
   #_w1 := "AlwaysTRUE" AND ("BUFF".PROCESS = 61);
   "IEC_Timer_0_DB_141".TON(IN := #_w1, PT := T#1s);
   IF "IEC_Timer_0_DB_141".Q AND ("IEC_Counter_0_DB_15".CV < "new"."BOW SET TIME"[3]) THEN
       "BUFF".PROCESS := 58;
   END_IF;
   "IEC_Counter_0_DB_15".CTU(CU := #_w1, R := "RESET_C15", PV := "new"."BOW SET TIME"[3]);
   #_w2 := "AlwaysTRUE" AND ("BUFF".PROCESS = 61) AND ("IEC_Counter_0_DB_15".CV >= "new"."BOW SET TIME"[3]);
   "IEC_Timer_0_DB_187".TON(IN := #_w2, PT := T#500MS);
   IF "IEC_Timer_0_DB_187".Q THEN
       "BUFF".PROCESS := 0;
       "CLOSURE ON" := TRUE;
       "IO BITS".HOOTER := TRUE;
   END_IF;
   "BOW DONE" := #_w2;
   IF #_w2 THEN "door2 allow" := TRUE; END_IF;
   "RESET_C15" := "BUFF".PROCESS = 0;
END_REGION
END_FUNCTION
